FUNCTION_BLOCK FB_Sequencer
VAR_INPUT
END_VAR
VAR_OUTPUT
END_VAR
VAR
END_VAR

END_FUNCTION_BLOCK

(* stored: Version 1.1.0.1
   POU FB_Sequencer: Id {082739e2-22b9-4029-95b6-33dd5a220750}, SpecialFunc None *)
